FUNCTION_BLOCK PY_MQTT_SUB (* Basic FB with empty ECC *)
  (* Standard: 61499-2 *)
  (* Version 1.0, 2024-12-03, obotnar *)
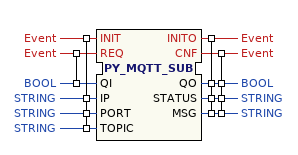
  EVENT_INPUT
    INIT WITH IP, PORT, TOPIC;
    REQ WITH QI;
  END_EVENT
  EVENT_OUTPUT
    INITO WITH STATUS, MSG, QO;
    CNF WITH STATUS, MSG, QO;
  END_EVENT
  VAR_INPUT
    QI : BOOL;
    IP : STRING;
    PORT : STRING;
    TOPIC : STRING;
  END_VAR
  VAR_OUTPUT
    QO : BOOL;
    STATUS : STRING;
    MSG : STRING;
  END_VAR
  EC_STATES
    START; (* Initial State *)
  END_STATES
END_FUNCTION_BLOCK
